TYPE TFTransportModuleStatus :
STRUCT
	Homed : BOOL; //Home modulo eseguito
	Error : UDINT;
	ErrorExtra : UDINT;
	PowerActive : BOOL; //Modulo in marcia
END_STRUCT
END_TYPE

(* stored: Version 1.1.0.1, ProductVersion 3.1.4024.11
   DUT TFTransportModuleStatus: Id {aeea829d-1601-4233-8b97-989d0097cc0a} *)
